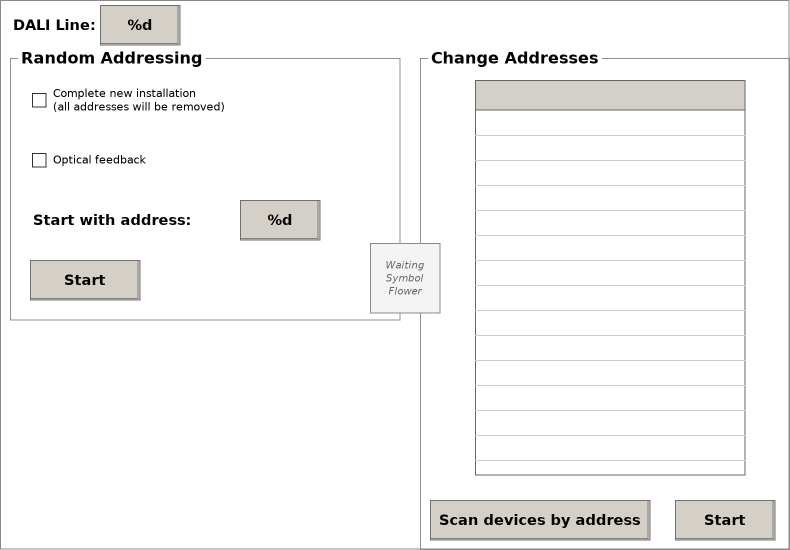
VISUALIZATION Visu_Part103Addressing  // 790x550
    GroupBox (420,50 370x500), "Change Addresses"
        Table (55,30 270x395), data array: DALI_Commissioning.fbPart103Addressing.aChangeAddressList
            p3854506369: DALI_Commissioning.fbPart103Addressing.aChangeAddressList[INDEX].nOldAddress
            p1892666644: DALI_Commissioning.fbPart103Addressing.aChangeAddressList[INDEX].nNewAddress
            p338671338: DALI_Commissioning.fbPart103Addressing.aChangeAddressList[INDEX].nRandomAddress
            p2170511999: DALI_Commissioning.fbPart103Addressing.aChangeAddressList[INDEX].nErrors
            Columns.Column.[0].Template: DALI_Commissioning.fbPart103Addressing.aNoShortAddress[INDEX]
            Columns.Column.[1].Template: DALI_Commissioning.fbPart103Addressing.aNoShortAddress[INDEX]; OnMouseClick: write the text variable via Default, min 0, max 63, title "New Short Address"
        Button (255,450 100x40), "Start"
            OnMouseClick: execute { DALI_Commissioning.fbPart103Addressing.bStartChangeAddress := TRUE; }
        Button (10,450 220x40), "Scan devices by address"
            OnMouseClick: execute { DALI_Commissioning.fbPart103Addressing.bScanDevices := TRUE; }
    GroupBox (10,50 390x270), "Random Addressing"
        Button (20,210 110x40), "Start"
            OnMouseClick: execute { DALI_Commissioning.fbPart103Addressing.bStartRandomAddressing := TRUE; }
        Checkbox (20,30 360x40), "Complete new installation (all addresses will be removed)", variable: DALI_Commissioning.fbPart103Addressing.bNewInstallation
        Checkbox (20,90 360x40), "Optical feedback", variable: DALI_Commissioning.fbPart103Addressing.bOpticalFeedback
        Textfield (20,150 200x40), "Start with address:"
        Button (230,150 80x40), "%d", text variable: DALI_Commissioning.fbPart103Addressing.nStartAddress
            OnMouseClick: write DALI_Commissioning.fbPart103Addressing.nStartAddress via Default, min 0, max 63, title "Insert Short Address"
    WaitingSymbolFlower (370,243 70x70), invisible if: DALI_Commissioning.fbPart103Addressing.bHideWaitSymbol
    Group (10,5 170x40)
        Textfield (0,0 110x40), "DALI Line:"
        Button (90,0 80x40), "%d", text variable: GVL_Internal.nDALILine
            OnMouseClick: write the text variable via Default, min 1, max 10, title "Choose line"
END_VISUALIZATION

(* stored: Version 1.1.0.1, ProductVersion 3.1.4024.9
   Visu Visu_Part103Addressing: Id {82d32c21-b584-4691-b14f-836230f5d6c2} *)
